INTERFACE I_Insertion2D

METHOD ABSTRACT align : BOOL
VAR_INPUT
	targetPos : REAL;
END_VAR
END_METHOD

PROPERTY Busy : BOOL
GET
END_GET
END_PROPERTY

PROPERTY Error : BOOL
GET
END_GET
END_PROPERTY

PROPERTY Home : BOOL
GET
END_GET
END_PROPERTY

METHOD ABSTRACT homingSequence : BOOL
VAR_INPUT
END_VAR
END_METHOD

METHOD ABSTRACT press : BOOL
VAR_INPUT
END_VAR
END_METHOD

METHOD ABSTRACT release : BOOL
VAR_INPUT
END_VAR
END_METHOD

METHOD ABSTRACT traverse : BOOL
VAR_INPUT
	direction : MC_Direction;
END_VAR
END_METHOD

END_INTERFACE

(* stored: Version 1.1.0.1, ProductVersion 3.1.4024.11
   Itf I_Insertion2D: Id {8e64ce60-22e0-4b91-ba46-fa91d2f7ae0e}
   Folder Properties: Id {a1c4999d-fc05-4f63-9c78-02da565e69f2}
   Method align: Id {fa643266-3d8f-4e66-aec5-e5710590bff8}
   Property Busy: Id {07cf4004-9de8-4cd7-9080-1436724591f2}
   Get Get: Id {3a58de26-60aa-46ff-a937-0baf2376a289}
   Property Error: Id {b4a0434b-ad4d-40cc-afba-ff64484c7904}
   Get Get: Id {ee0b8ff1-e35f-48bd-83b4-e127e7f01aa1}
   Property Home: Id {567b309e-9957-4d04-acb9-a5e56d9c7992}
   Get Get: Id {5e81f538-0161-431e-b40d-1900836e48be}
   Method homingSequence: Id {e50d8f3c-3832-479d-9ea8-d077b3535f03}
   Method press: Id {d84955f1-e0a2-4a22-92a7-c7477ef94736}
   Method release: Id {92bdeeca-e13f-4d7f-bf24-c4aad1f47945}
   Method traverse: Id {62c2b24a-3291-4b2f-ac0b-b5af5509b392} *)
